{attribute addProperty BoxType "EL1262-0000-0002"}
{attribute addProperty Id "Ch2_CycleCountAT %I*UINT162"}
{attribute addProperty CRC "2104859732"}
{attribute addProperty SizeInBites "16"}
{attribute addProperty SizeInBytes "2"}
TYPE Ch2_CycleCount_7D759C54 :
STRUCT
	{attribute addProperty Name "Ch2_CycleCount"}
	Ch2_CycleCount AT %I* : UINT;
END_STRUCT
END_TYPE

(* stored: Version 1.2.0.0, ProductVersion 3.1.4024.9
   DUT Ch2_CycleCount_7D759C54: Id {495d8c2d-ae82-4d33-aac3-c83f39c7b788} *)
